TYPE ST_Bel_Lampen_Monitoring :
STRUCT
	Betrieb	: BOOL;
	Relative_Leistung	: REAL;
END_STRUCT
END_TYPE

(* stored: Version 1.1.0.1, ProductVersion 3.1.4024.9
   DUT ST_Bel_Lampen_Monitoring: Id {8b6ad693-b45b-47be-a7a4-093ee3b2cd7e} *)
